// TIA Portal project "Sırayla Paket Dağıtma" (V15)
// Vorlageprojekt für das Buch mit Zielsystem S7-1200

(* hardware
DEVICE "S7-1200-Station_1"  S7-1200 Station
   slot 0: "Baugruppenträger_0"  Rack  V1.0
   slot 1: "PLC_1"  CPU 1211C DC/DC/DC  6ES7 211-1AE40-0XB0  V4.1
*)

// ===== PLC "PLC_1"  CPU 1211C DC/DC/DC =====

VAR_GLOBAL   // PLC tag table "Standard-Variablentabelle"
   "Sensör" AT %I0.5 : Bool;
   "Reset Button" AT %I0.4 : Bool;
   "Start" AT %I0.0 : Bool;
   "Konveyor_1" AT %Q0.0 : Bool;
   "Konveyor_2" AT %Q0.1 : Bool;
   "Stop_Button" AT %I0.1 : Bool;
   "Sayma_Değeri" AT %QW30 : Int;
   "KOL_3" AT %Q0.2 : Bool;
   "Kayış_3" AT %Q0.3 : Bool;
   "Kol_2" AT %Q0.4 : Bool;
   "Kayış_2" AT %Q0.5 : Bool;
   "Tag_1" AT %Q0.6 : Bool;
   "Tag_2" AT %Q0.7 : Bool;
   "Sensör Lambası" AT %Q1.0 : Bool;
   "Tepe lambası" AT %Q1.1 : Bool;
   "Tag_3" AT %Q1.2 : Bool;
END_VAR

// folder: System blocks/Program resources

DATA_BLOCK "Sayıcı"   // DB5
{ S7_Optimized_Access := 'TRUE' }
AUTHOR : Simatic
FAMILY : IEC
NAME : CNTR
VERSION : 1.0
// stored: InstanceOfName IEC_COUNTER
"IEC_COUNTER"
BEGIN
END_DATA_BLOCK

// folder: (top level)

FUNCTION "MHJ-PLC-Lab-Function-S71200" : Void   // FC9000, SCL
{ S7_Optimized_Access := 'TRUE' }
VERSION : 0.1
   VAR_TEMP
      rdTimeReturn : Int;
      outputTime : DTL;
      SyncVal : Byte;
      forVal : Int;
      forVal_2 : Int;
      Value : Byte;
   END_VAR
   VAR CONSTANT
      CompVal : Byte := 16#34;
      Value_01 : Byte := 16#11;
      Value_01_DW : DWord := 16#A165_D992;
      Value_02_DW : DWord := 16#58BE_4401;
   END_VAR
BEGIN

   #Value:=PEEK(area := 16#82,
        dbNumber := 0,
        byteOffset := 511);
   #Value := #Value + 1;

   POKE(area := 16#82,
        dbNumber := 0,
        byteOffset := 511,
        value := #Value);

   POKE(area:=16#81,
        dbNumber:=0,
        byteOffset:=1016,
        value:=#Value_01_DW);
   POKE(area := 16#81,
        dbNumber := 0,
        byteOffset := 1020,
        value := #Value_02_DW);

   POKE(area := 16#81,
        dbNumber := 0,
        byteOffset := 511,
        value := B#16#00);

   FOR #forVal := 0 TO 120 DO
       FOR #forVal_2:=0 TO 10 DO
           #rdTimeReturn:=RD_SYS_T(#outputTime);
           #rdTimeReturn := WR_SYS_T(#outputTime);
           #rdTimeReturn := RD_SYS_T(#outputTime);
           #rdTimeReturn := WR_SYS_T(#outputTime);
       END_FOR;
       #SyncVal:= PEEK(area := 16#81,
                      dbNumber := 0,
                      byteOffset := 511);
       IF #SyncVal = #CompVal THEN
          GOTO M_1;
       END_IF;
   END_FOR;
   RETURN;

   M_1:
   POKE(area := 16#81,
        dbNumber := 0,
        byteOffset := 511,
        value := B#16#0);
END_FUNCTION

ORGANIZATION_BLOCK "Main"   // OB1, LAD, ProgramCycle
TITLE = "Main Program Sweep (Cycle)"
{ S7_Optimized_Access := 'TRUE' }
VERSION : 0.1
   VAR_INPUT
      Initial_Call : Bool;   // Initial call of this OB
      Remanence : Bool;   // =True, if remanent data are available
   END_VAR
BEGIN

REGION Network 1: Konnektierungsbaustein für PLC-Lab
   // Im Netzwerk 1 wird der Konnektierungsbaustein für PLC-Lab aufgerufen.
   // Dieser Aufruf darf nicht entfernt werden!
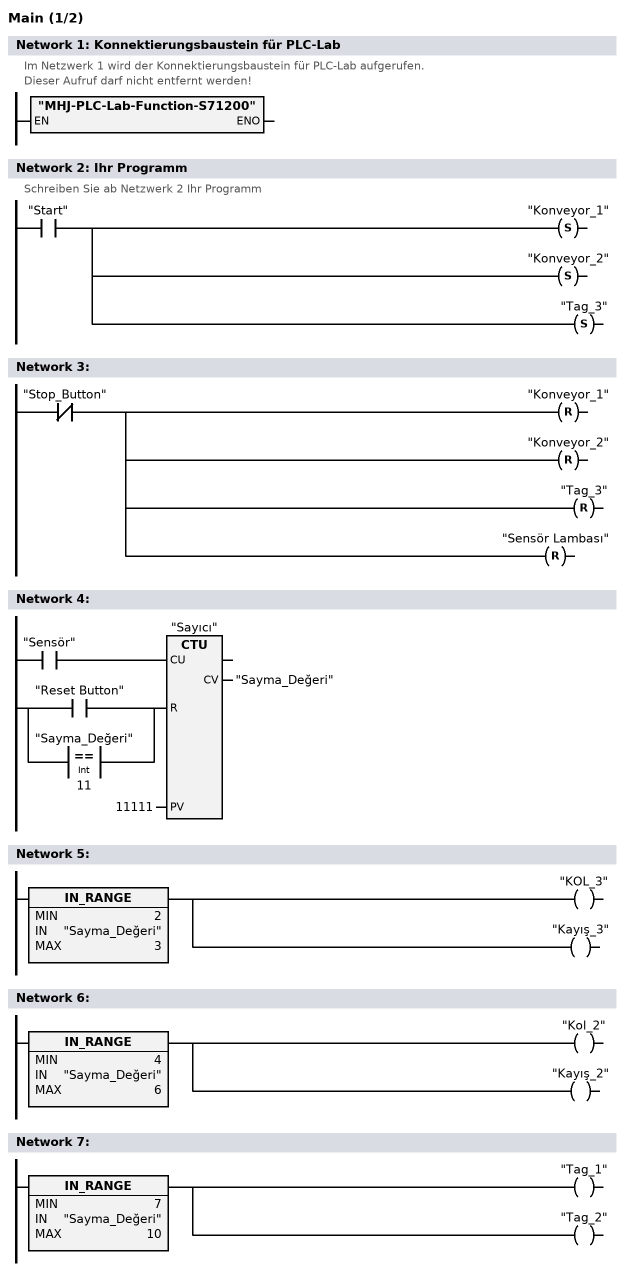
   RUNG wire#powerrail
      "MHJ-PLC-Lab-Function-S71200"()
   END_RUNG
   // the same network as SCL:
   "MHJ-PLC-Lab-Function-S71200"();
END_REGION

REGION Network 2: Ihr Programm
   // Schreiben Sie ab Netzwerk 2 Ihr Programm
   RUNG wire#powerrail
      Contact( "Start" )
      wire#w1
      S_Coil( "Konveyor_1" )
   END_RUNG
   RUNG wire#w1
      S_Coil( "Konveyor_2" )
   END_RUNG
   RUNG wire#w1
      S_Coil( "Tag_3" )
   END_RUNG
   // the same network as SCL:
   IF "Start" THEN
       "Konveyor_1" := TRUE;
       "Konveyor_2" := TRUE;
       "Tag_3" := TRUE;
   END_IF;
END_REGION

REGION Network 3
   RUNG wire#powerrail
      I_Contact( "Stop_Button" )
      wire#w1
      R_Coil( "Konveyor_1" )
   END_RUNG
   RUNG wire#w1
      R_Coil( "Konveyor_2" )
   END_RUNG
   RUNG wire#w1
      R_Coil( "Tag_3" )
   END_RUNG
   RUNG wire#w1
      R_Coil( "Sensör Lambası" )
   END_RUNG
   // the same network as SCL:
   IF NOT "Stop_Button" THEN
       "Konveyor_1" := FALSE;
       "Konveyor_2" := FALSE;
       "Tag_3" := FALSE;
       "Sensör Lambası" := FALSE;
   END_IF;
END_REGION

REGION Network 4
   "Sayıcı".CTU(CU := "Sensör", R := "Reset Button" OR ("Sayma_Değeri" = 11), PV := 11111, CV => "Sayma_Değeri");
END_REGION

REGION Network 5
   RUNG wire#powerrail
      { S7_Templates := "SrcType := Int" } InRange(min := 2, in := "Sayma_Değeri", max := 3)
      wire#w1
      Coil( "KOL_3" )
   END_RUNG
   RUNG wire#w1
      Coil( "Kayış_3" )
   END_RUNG
   // the same network as SCL:
   "KOL_3" := (2 <= "Sayma_Değeri") AND ("Sayma_Değeri" <= 3);
   "Kayış_3" := "KOL_3";
END_REGION

REGION Network 6
   RUNG wire#powerrail
      { S7_Templates := "SrcType := Int" } InRange(min := 4, in := "Sayma_Değeri", max := 6)
      wire#w1
      Coil( "Kol_2" )
   END_RUNG
   RUNG wire#w1
      Coil( "Kayış_2" )
   END_RUNG
   // the same network as SCL:
   "Kol_2" := (4 <= "Sayma_Değeri") AND ("Sayma_Değeri" <= 6);
   "Kayış_2" := "Kol_2";
END_REGION

REGION Network 7
   RUNG wire#powerrail
      { S7_Templates := "SrcType := Int" } InRange(min := 7, in := "Sayma_Değeri", max := 10)
      wire#w1
      Coil( "Tag_1" )
   END_RUNG
   RUNG wire#w1
      Coil( "Tag_2" )
   END_RUNG
   // the same network as SCL:
   "Tag_1" := (7 <= "Sayma_Değeri") AND ("Sayma_Değeri" <= 10);
   "Tag_2" := "Tag_1";
END_REGION

REGION Network 8
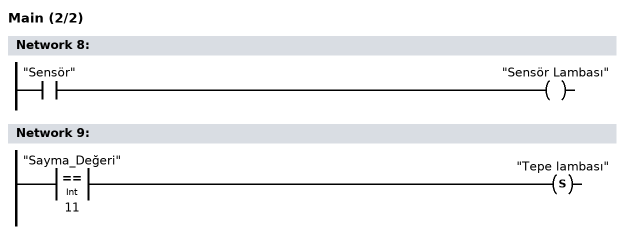
   RUNG wire#powerrail
      Contact( "Sensör" )
      Coil( "Sensör Lambası" )
   END_RUNG
   // the same network as SCL:
   "Sensör Lambası" := "Sensör";
END_REGION

REGION Network 9
   RUNG wire#powerrail
      { S7_Templates := "SrcType := Int" } EQ_Contact(in1 := "Sayma_Değeri", in2 := 11)
      S_Coil( "Tepe lambası" )
   END_RUNG
   // the same network as SCL:
   IF "Sayma_Değeri" = 11 THEN "Tepe lambası" := TRUE; END_IF;
END_REGION
END_ORGANIZATION_BLOCK